PROGRAM ReadWriteOPCvariables
VAR
END_VAR


GVL_OPC.OPC_ReactorTemperature := GVL_IO.reactorTemperatureUpper;
GVL_OPC.OPC_TemperatureContactor := GVL_IO.reactorTemperatureContactor;
GVL_OPC.OPC_ReactorPressure := ReactorLevelAndPressureController.iPressureScaledValue;//ReactorLevelAndPressureControl.iPressureScaledValue;
IF ReactorTemperatureController._autoControlSelected THEN//ReactorTemperatureControl.bTempCon THEN
	GVL_OPC.OPC_ReactorTemperatureSetpoint := REAL_TO_INT(ReactorTemperatureController._temperatureSetpoint);//REAL_TO_INT(ReactorTemperatureControl.iTemperatureSetpoint);
ELSE
	GVL_OPC.OPC_ReactorTemperatureSetpoint := 0;
END_IF
GVL_OPC.OPC_SlurryInletValve := GVL_IO.reactorInletValve;
GVL_OPC.OPC_SlurryOutletValve := GVL_IO.reactorOutletValve;

GVL_OPC.OPC_CO2VolumetricFlow := SerialCommunicationHandler.flowMeasurement;
GVL_OPC.OPC_PumpingPressure := SerialCommunicationHandler.pumpingPressureMeasurement;
GVL_OPC.OPC_PumpingPressureSetpoint := SerialCommunicationHandler.pumpingPressureSetpoint;
GVL_OPC.OPC_PreHeaterTemperature := SerialCommunicationHandler.preHeaterTemperatureMeasurement;
GVL_OPC.OPC_PreHeaterTemperatureSetpoint := SerialCommunicationHandler.preHeaterTemperatureSetpoint;
GVL_OPC.OPC_SeparatorTemperature := SerialCommunicationHandler.separatorTemperatureMeasurement;
GVL_OPC.OPC_SeparatorTemperatureSetpoint := SerialCommunicationHandler.separatorTemperatureSetpoint;

END_PROGRAM

(* stored: Version 1.1.0.1, ProductVersion 3.1.4024.9
   POU ReadWriteOPCvariables: Id {f3380c8e-c00f-42bf-a0c6-face89438324}, SpecialFunc None *)
